{attribute 'qualified_only'}
{attribute 'strict'}
{attribute 'to_string'}
TYPE E_ManuelModes :
(
	ManDirect,
	ManConst,
	ManSpeed
);
END_TYPE

(* stored: Version 1.1.0.1
   DUT E_ManuelModes: Id {407ff541-c4fa-43f5-89ee-e1ad4ea53de1} *)
